FUNCTION_BLOCK Seq_2
VAR_INPUT
	// Basis-Inputs
	bExecute			:BOOL;				// Trigger für Ausführung von Sequenz
	iSysCommand			:eSystemCommand;	// Steuerungsvariabel von System (Resetten)
	
	// Prozess-Inputs 
	Position_1			:sRoboterProzessVariablen;
	Position_2			:sRoboterProzessVariablen;
	Position_3			:sRoboterProzessVariablen;
	
END_VAR
VAR_OUTPUT
	bDone				:BOOL;				// Information ob Sequenz ausgfeührt wurde
	bBusy				:BOOL;				// Information ob Sequenz im Moment ausgeführt wird
	bError				:BOOL;				// Information ob sich Sequenz in Fehlerzustand befindet
END_VAR
VAR
	// Sequenz-Zustände
	iState				:eSequenceState;
	
	// Startvariablen (FB soll nur bei einer steigenden Flanke gestartet werden)
	fTrigger			:R_TRIG;			// Erkennung einer steigenden Flanke für den Starte
	fSwitch				:SR;				// Setzen des Signals
	bSwitchResett		:BOOL;				// Resetten des Signals
	
	// Zustandsvariablen
	bStarten			:BOOL;
	bStoppen			:BOOL;
	bResetten			:BOOL;
	
	// Management-Variablen:
	bFinished			:BOOL;
	bInit				:BOOL;
	
	// Skill-Instanziierungen
	P2P_Movement		:Skill_Position_anfahren_erweitert;
	Position			:sRoboterProzessVariablen;
END_VAR

// Aufrufen von Skills und Ablauf
Ablauf();	
Skills();

//_______________________________________________________________
// Reaktion auf Fehler
IF bError THEN
	iState := 3;
END_IF	

// Reaktion auf Input-Variablen: 
	// Starten
	fTrigger(CLK := bExecute);
	fSwitch(Set1 := fTrigger.Q);
	
	IF fSwitch.Q1 THEN
		bStarten := TRUE;
	ELSE
		bStarten := FALSE;
	END_IF
	
	// Stoppen
	IF iSysCommand = 3 THEN
		bStoppen := TRUE;	
	ELSE 
		bStoppen := FALSE;	
	END_IF
	
	// Stoppen
	IF iSysCommand = 4 THEN
		bResetten := TRUE;	
	ELSE 
		bResetten := FALSE;	
	END_IF



//_______________________________________________________________
// Zustandsmanagement
CASE iState OF 
	0:	// BEREIT
			// DO	
			fSwitch.RESET := FALSE;
				
			// TRANSITION
			IF bStarten THEN
				fSwitch.RESET := TRUE;
				iState := 1;																							// Starten des Objektes 
			END_IF
	// ________________________________________________________________________________			
	1:	// LAUFEND
			// DO
			bBusy := TRUE;	

			IF bStoppen THEN
				SFCReset := TRUE;
				bBusy := FALSE;
			END_IF	
			
			// TRANSITION
			IF bFinished THEN
				bFinished := FALSE;
				bBusy := FALSE;
				iState := 2;
			END_IF
			
			IF bInit THEN
				bInit := FALSE;
				SFCReset := FALSE;
				iState := 0;
			END_IF

	// ________________________________________________________________________________					
	2:	// ABGESCHLOSSEN
			// DO
			bDone := TRUE;			
						
			// TRANSITION
			IF bDone THEN
				bDone := FALSE;
				iState := 0;
			END_IF
	// ________________________________________________________________________________					
	3:	// FEHLER
			// DO
			bDone := FALSE;
			bBusy := FALSE;
			
			// TRANSITION
			IF bResetten THEN
				bError := FALSE;
				iState := 0;
			END_IF
			
END_CASE

ACTION Ablauf:
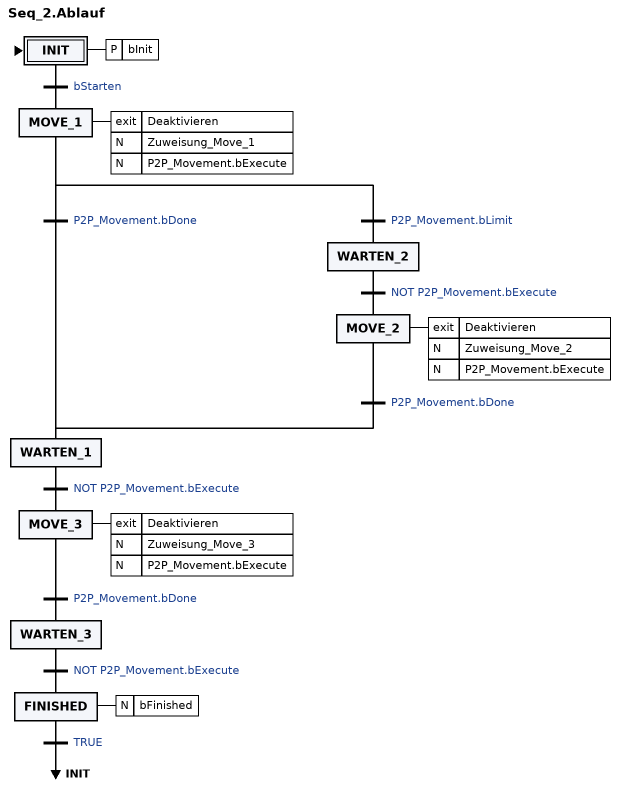
INITIAL_STEP INIT:
    bInit(P);
END_STEP
TRANSITION FROM INIT TO MOVE_1
    := bStarten;
END_TRANSITION
STEP MOVE_1:
    Deaktivieren(P0);  // exit action
    Zuweisung_Move_1(N);
    P2P_Movement.bExecute(N);
END_STEP
TRANSITION FROM MOVE_1 TO WARTEN_1
    := P2P_Movement.bDone;
END_TRANSITION
TRANSITION FROM MOVE_1 TO WARTEN_2
    := P2P_Movement.bLimit;
END_TRANSITION
STEP WARTEN_2:
END_STEP
TRANSITION FROM WARTEN_2 TO MOVE_2
    := NOT P2P_Movement.bExecute;
END_TRANSITION
STEP MOVE_2:
    Deaktivieren(P0);  // exit action
    Zuweisung_Move_2(N);
    P2P_Movement.bExecute(N);
END_STEP
TRANSITION FROM MOVE_2 TO WARTEN_1
    := P2P_Movement.bDone;
END_TRANSITION
STEP WARTEN_1:
END_STEP
TRANSITION FROM WARTEN_1 TO MOVE_3
    := NOT P2P_Movement.bExecute;
END_TRANSITION
STEP MOVE_3:
    Deaktivieren(P0);  // exit action
    Zuweisung_Move_3(N);
    P2P_Movement.bExecute(N);
END_STEP
TRANSITION FROM MOVE_3 TO WARTEN_3
    := P2P_Movement.bDone;
END_TRANSITION
STEP WARTEN_3:
END_STEP
TRANSITION FROM WARTEN_3 TO FINISHED
    := NOT P2P_Movement.bExecute;
END_TRANSITION
STEP FINISHED:
    bFinished(N);
END_STEP
TRANSITION FROM FINISHED TO INIT
    := TRUE;
END_TRANSITION
// branch label Branch0_Ablauf
END_ACTION

ACTION Deaktivieren:
P2P_Movement.bExecute := FALSE;
END_ACTION

ACTION Skills:
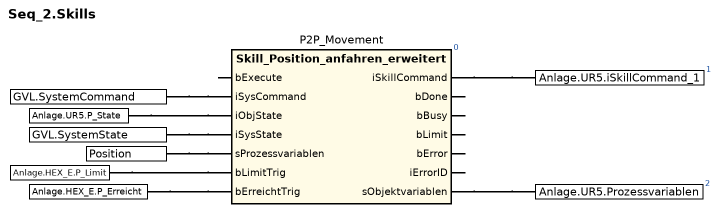
P2P_Movement(
    iSysCommand := GVL.SystemCommand,
    iObjState := Anlage.UR5.P_State,
    iSysState := GVL.SystemState,
    sProzessvariablen := Position,
    bLimitTrig := Anlage.HEX_E.P_Limit,
    bErreichtTrig := Anlage.HEX_E.P_Erreicht); // Skill_Position_anfahren_erweitert
Anlage.UR5.iSkillCommand_1 := P2P_Movement.iSkillCommand;
Anlage.UR5.Prozessvariablen := P2P_Movement.sObjektvariablen;
END_ACTION

ACTION Zuweisung_Move_1:
Position := Position_1;
END_ACTION

ACTION Zuweisung_Move_2:
Position := Position_2;
END_ACTION

ACTION Zuweisung_Move_3:
Position := Position_3;
END_ACTION

END_FUNCTION_BLOCK

(* stored: Version 1.1.0.1
   POU Seq_2: Id {3bc0ea8d-9b53-40dd-bf05-3b837e1df7f5}, SpecialFunc None
   Folder 00_Hilfsaktionen: Id {4afbbfdd-129c-46f2-872e-b5fb2541c591}
   Folder 01_Zuweisung: Id {4ce987ba-19ee-4bd0-bd13-960767bd0fa7}
   Action Ablauf: Id {76d518a6-c73e-4a80-9596-7ebebe4d8963}
   Action Deaktivieren: Id {da903ee6-8ef9-438e-94c2-476a7cd631f9}
   Action Skills: Id {1e66b983-0e15-4e6d-bc59-87a209a17d2c}
   Action Zuweisung_Move_1: Id {ab95cd4b-8382-40dc-ba8e-e0b0a2ad4347}
   Action Zuweisung_Move_2: Id {5500c7de-505c-4e5a-9b56-7ee209ad5737}
   Action Zuweisung_Move_3: Id {aa31d0cc-727e-4508-914d-8168c114c355} *)
